Universal Robots PolyScope program: Hospital_base.urp

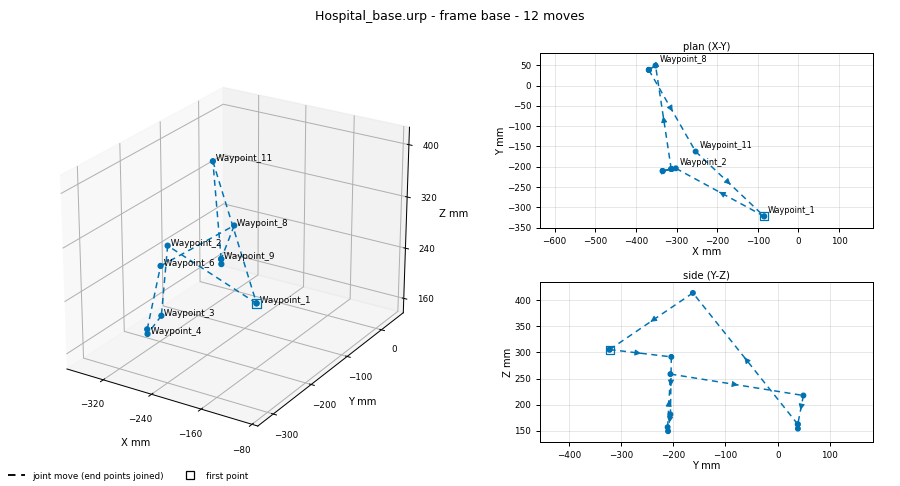
[picture p0: tool path of Hospital_base.urp in frame base, 12 of 12 moves have a stored position in this frame; points joined in program order, loops and branches not executed]
Program Hospital_base (installation=default directory=/programs/usbdisk/Zahra1 createdIn=5.11.11.1010533 lastSavedIn=5.11.11.1010533 robotSerialNumber=20205300864)
Calibrated DH parameters: a=[-0.000166, -0.243494, -0.153108, 0.000057, -0.000123, 0]; d=[0.151897, -1.34267, 53.988124, -52.514559, 0.085283, 0.092193]; alpha=[1.572472, -0.003756, 0.002824, 1.570807, -1.572621, 0]; deltaTheta=[0, 0.020704, 7.033215, -0.770746, 0.000004, 0]
Robot Program (runOnlyOnce=true)
  MoveJ speed 60 deg/s, acceleration 80 deg/s^2 (useActiveTCP=true) feature=Base
    Waypoint Waypoint_1: TCP in base x=-84.309 y=-321.871 z=305.49 mm, rx=-2.081 ry=-2.2572 rz=0.0985 rad; joints [-79.979, -91.199, -87.973, -91.697, 84.67, 815.506] deg
    URCap Gripper Activate (Robotiq_Grippers, Robotiq Inc.) dataModel(ResetAndActivateKey=false)
    URCap Gripper (Robotiq_Grippers, Robotiq Inc.) dataModel(position=0.0, force=100.0, speed=100.0, positionInDouble=0.0, forceInDouble=100.0, speedInDouble=100.0, slaveIds=[9], blocking=true, robotCompliant=false)
    Waypoint Waypoint_2: TCP in base x=-301.766 y=-203.688 z=291.505 mm, rx=-2.1508 ry=-2.1871 rz=0.1194 rad; joints [-123.668, -97.785, -86.402, -82.106, 85.116, 775.322] deg
    Waypoint Waypoint_3: TCP in base x=-313.016 y=-205.394 z=181.365 mm, rx=-2.1426 ry=-2.2429 rz=0.1036 rad; joints [-125.681, -108.779, -103.688, -53.947, 87.3, 771.785] deg
    Waypoint Waypoint_4: TCP in base x=-334.126 y=-209.928 z=149.191 mm, rx=2.2019 ry=2.2181 rz=0.0349 rad; joints [-128.87, -118.285, -97.038, -55.749, 91.012, 770.871] deg
    URCap Gripper (Robotiq_Grippers, Robotiq Inc.) dataModel(position=48.23529411764706, force=80.0, speed=70.0, positionInDouble=48.23529411764706, forceInDouble=80.0, speedInDouble=70.0, slaveIds=[9], blocking=true, robotCompliant=true)
    Waypoint Waypoint_5: motionParameters(jointSpeed=0.698132 jointAcceleration=0.698132 cartesianSpeed=0.25 cartesianAcceleration=1.2); TCP in base x=-334.014 y=-210.731 z=156.871 mm, rx=2.2024 ry=2.2182 rz=0.0357 rad; joints [-128.771, -117.33, -96.101, -57.668, 90.994, 770.974] deg
    Waypoint Waypoint_6: TCP in base x=-313.009 y=-205.387 z=258.545 mm, rx=-2.1427 ry=-2.2429 rz=0.1033 rad; joints [-125.652, -101.83, -90.39, -74.205, 87.307, 771.769] deg
    Waypoint Waypoint_8: TCP in base x=-351.594 y=49.204 z=217.576 mm, rx=3.1263 ry=0.0123 rz=-0.0104 rad; joints [-166.661, -101.222, -101.412, -66.689, 90.779, 823.048] deg
    Waypoint Waypoint_9: TCP in base x=-368.154 y=38.457 z=162.457 mm, rx=-3.1173 ry=0.0205 rz=-0.0327 rad; joints [-165.115, -111.176, -103.789, -56.457, 88.981, 825.829] deg
    Waypoint Waypoint_12: motionParameters(jointSpeed=0.349066 jointAcceleration=0.174533 cartesianSpeed=0.25 cartesianAcceleration=1.2); TCP in base x=-367.97 y=38.67 z=154.073 mm, rx=-3.1173 ry=0.0206 rz=-0.0327 rad; joints [-165.144, -112.338, -104.802, -54.28, 88.978, 825.808] deg
    URCap Gripper (Robotiq_Grippers, Robotiq Inc.) dataModel(position=23.52941176470588, force=70.0, speed=41.0, positionInDouble=23.52941176470588, forceInDouble=70.0, speedInDouble=41.0, slaveIds=[9], blocking=true, robotCompliant=true)
    Waypoint Waypoint_9: TCP in base x=-368.154 y=38.457 z=162.457 mm, rx=-3.1173 ry=0.0205 rz=-0.0327 rad; joints [-165.115, -111.176, -103.789, -56.457, 88.981, 825.829] deg
    Waypoint Waypoint_11: TCP in base x=-252.972 y=-162.386 z=413.928 mm, rx=2.8045 ry=0.6128 rz=-0.121 rad; joints [-124.146, -84.485, -71.424, -99.818, 97.741, 842.242] deg
    Waypoint Waypoint_1: TCP in base x=-84.309 y=-321.871 z=305.49 mm, rx=-2.081 ry=-2.2572 rz=0.0985 rad; joints [-79.979, -91.199, -87.973, -91.697, 84.67, 815.506] deg
